TYPE mmHg :
STRUCT
    _ : REAL;
    unit : STRING := 'mmHg';
END_STRUCT
END_TYPE

(* stored: Version 1.1.0.1, ProductVersion 3.1.4024.4
   DUT mmHg: Id {4cee1e1f-3465-4a38-afd1-e11c447626ed} *)
